FUNCTION_BLOCK Event_Listener EXTENDS FB_ListenerBase
VAR_INPUT
END_VAR
VAR_OUTPUT
END_VAR
VAR
	sJsonAttribute : STRING (10000);	
	hr : HRESULT;
	
	nCntMessagesSent : INT;
	nCntAlarmsRaised : INT;
	nCntAlarmsConfirmed : INT;
	nCntAlarmsCleared : INT;
	
	//text retrieval of message
	fbRequestEventText : FB_RequestEventText;
	{attribute 'TcEncoding':='UTF-8'}
	sLastMessageText : STRING;
	bReqText : BOOL;
END_VAR

METHOD Execute : HRESULT
VAR_INPUT
END_VAR
Execute := SUPER^.Execute(); //retrieve events

//retrieve the text of a message
IF 	bReqText AND fbRequestEventText.bError THEN 
	sLastMessageText := 'Error';
	bReqText := FALSE; 
ELSIF bReqText AND NOT  fbRequestEventText.bBusy THEN
	fbRequestEventText.GetString(sLastMessageText, SIZEOF(sLastMessageText));
	bReqText := FALSE;
END_IF
END_METHOD

METHOD OnAlarmCleared
VAR_INPUT
	fbEvent : REFERENCE TO FB_TcEvent;
END_VAR
nCntAlarmsCleared := nCntAlarmsCleared + 1;
END_METHOD

METHOD OnAlarmConfirmed
VAR_INPUT
	fbEvent : REFERENCE TO FB_TcEvent;
END_VAR
nCntAlarmsConfirmed := nCntAlarmsConfirmed + 1;
fbEvent;
END_METHOD

METHOD OnAlarmRaised
VAR_INPUT
	fbEvent: REFERENCE TO FB_TcEvent;
END_VAR
VAR
	str1 : STRING;
	str2 : STRING := 'My custom source';
END_VAR
hr := fbEvent.GetJsonAttribute(sJsonAttribute, SIZEOF(sJsonAttribute));
nCntAlarmsRaised := nCntAlarmsRaised + 1;
//IF fbEvent.EqualsTo(TC_Events.MyEventClass.MySecondAlarm) THEN
	// Event that got raised is my 2nd alarm
//END_IF

str1 := fbEvent.ipSourceInfo.sName;
IF str1 = str2 THEN
	// This is my even source
END_IF
END_METHOD

METHOD OnMessageSent
VAR_INPUT
	fbEvent : REFERENCE TO FB_TcEvent;
END_VAR
hr := fbEvent.GetJsonAttribute(sJsonAttribute, SIZEOF(sJsonAttribute));
nCntMessagesSent := nCntMessagesSent + 1;

fbRequestEventText.Request(eventClass:=fbEvent.EventClass, nEventId:=fbEvent.nEventId, nLangId:=1033, ipArgs:=fbEvent.ipArguments );
bReqText := TRUE;
END_METHOD

END_FUNCTION_BLOCK

(* stored: Version 1.1.0.1, ProductVersion 3.1.4022.16
   POU Event_Listener: Id {557c767d-437c-4e1b-8ea2-0e28629919b1}, SpecialFunc None
   Method Execute: Id {39f9c2a5-ab39-4546-be43-6992f41e147b}
   Method OnAlarmCleared: Id {e597da0e-0e69-4914-9fca-7e402a2c6aa9}
   Method OnAlarmConfirmed: Id {9ef40bd9-c98c-419d-b6db-2b02aa1c32e3}
   Method OnAlarmRaised: Id {c2f0f5b8-0a93-43bf-a7d0-bbe70b0c3004}
   Method OnMessageSent: Id {7c9f4a3c-e1ee-4422-97be-64623f192bb9} *)
